// TIA Portal V21 export
TYPE "coneCrusherSta"
   STRUCT
      status : Struct
         ready : Bool;
         operation : Bool;
         run : Bool;
         alm : Bool;
         unackAlm : Bool;
         premoldingSw : Bool;
         prestartAlmOn : Bool;
         prestartAlmFb : Bool;
         prestartAlmFalseFb : Bool;
         prestartAlmNoFb : Bool;
         feedEn : Bool;
      END_STRUCT;
      statusDWord : DWord;
      "step" : USInt;
      stepTime : LTime;
      alm : "coneCrusherAlm";
      almDWord { S7_SetPoint := 'True'} : DWord;
      StopCtx : "coneCrusherStopCtx";
   END_STRUCT;
END_TYPE
